FUNCTION BoolVariableArrayToInteger : LINT;
VAR_IN_OUT
	arr : POINTER TO BOOL;
END_VAR
VAR
	i : DINT;
	j : DINT;
END_VAR

//FOR i:=numElements TO 0 BY -1 DO
FOR i:=UPPER_BOUND(arr, 1) TO LOWER_BOUND(arr, 1) BY -1 DO
	IF j < SIZEOF(BoolVariableArrayToInteger) * 8 THEN
		
		BoolVariableArrayToInteger.0 := arr[i];		
		IF i <> LOWER_BOUND(arr, 1) THEN
			BoolPointerArrayToInteger := SHL(BoolVariableArrayToInteger, 1);
		END_IF
		
	END_IF
	
	j := j + 1;
END_FOR

END_FUNCTION

(* stored: Version 1.1.0.1, ProductVersion 3.1.4024.11
   POU BoolVariableArrayToInteger: Id {9d36b047-c6f5-4988-8250-82848c033c4d}, SpecialFunc None *)
